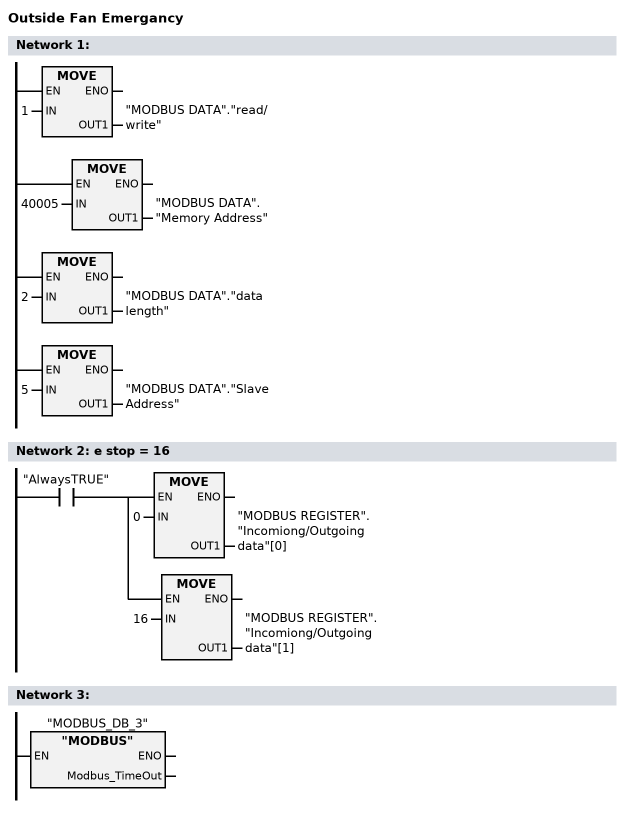
   RUNG wire#powerrail
      Move(in := 1, out1 => "MODBUS DATA"."read/write")
   END_RUNG
   RUNG wire#powerrail
      Move(in := 40005, out1 => "MODBUS DATA"."Memory Address")
   END_RUNG
   RUNG wire#powerrail
      Move(in := 2, out1 => "MODBUS DATA"."data length")
   END_RUNG
   RUNG wire#powerrail
      Move(in := 5, out1 => "MODBUS DATA"."Slave Address")
   END_RUNG
   // the same network as SCL:
   "MODBUS DATA"."read/write" := 1;
   "MODBUS DATA"."Memory Address" := 40005;
   "MODBUS DATA"."data length" := 2;
   "MODBUS DATA"."Slave Address" := 5;
END_REGION

REGION Network 2: e stop = 16
   RUNG wire#powerrail
      Contact( "AlwaysTRUE" )
      wire#w1
      Move(in := 0, out1 => "MODBUS REGISTER"."Incomiong/Outgoing data"[0])
   END_RUNG
   RUNG wire#w1
      Move(in := 16, out1 => "MODBUS REGISTER"."Incomiong/Outgoing data"[1])
   END_RUNG
   // the same network as SCL:
   IF "AlwaysTRUE" THEN
       "MODBUS REGISTER"."Incomiong/Outgoing data"[0] := 0;
       "MODBUS REGISTER"."Incomiong/Outgoing data"[1] := 16;
   END_IF;
END_REGION

REGION Network 3
   RUNG wire#powerrail
      "MODBUS_DB_3"(Modbus_TimeOut =>)
   END_RUNG
   // the same network as SCL:
   "MODBUS_DB_3"();   // "MODBUS"
END_REGION
END_FUNCTION_BLOCK

FUNCTION_BLOCK "Inside Fan Emergancy"   // FB22, LAD
{ S7_Optimized_Access := 'TRUE' }
VERSION : 0.1
BEGIN

REGION Network 1
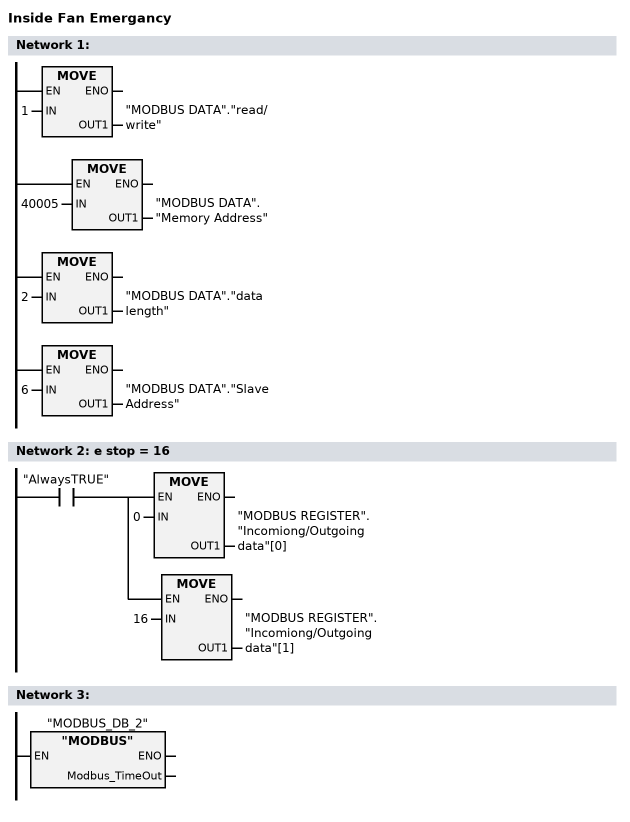
   RUNG wire#powerrail
      Move(in := 1, out1 => "MODBUS DATA"."read/write")
   END_RUNG
   RUNG wire#powerrail
      Move(in := 40005, out1 => "MODBUS DATA"."Memory Address")
   END_RUNG
   RUNG wire#powerrail
      Move(in := 2, out1 => "MODBUS DATA"."data length")
   END_RUNG
   RUNG wire#powerrail
      Move(in := 6, out1 => "MODBUS DATA"."Slave Address")
   END_RUNG
   // the same network as SCL:
   "MODBUS DATA"."read/write" := 1;
   "MODBUS DATA"."Memory Address" := 40005;
   "MODBUS DATA"."data length" := 2;
   "MODBUS DATA"."Slave Address" := 6;
END_REGION

REGION Network 2: e stop = 16
   RUNG wire#powerrail
      Contact( "AlwaysTRUE" )
      wire#w1
      Move(in := 0, out1 => "MODBUS REGISTER"."Incomiong/Outgoing data"[0])
   END_RUNG
   RUNG wire#w1
      Move(in := 16, out1 => "MODBUS REGISTER"."Incomiong/Outgoing data"[1])
   END_RUNG
   // the same network as SCL:
   IF "AlwaysTRUE" THEN
       "MODBUS REGISTER"."Incomiong/Outgoing data"[0] := 0;
       "MODBUS REGISTER"."Incomiong/Outgoing data"[1] := 16;
   END_IF;
END_REGION

REGION Network 3
   RUNG wire#powerrail
      "MODBUS_DB_2"(Modbus_TimeOut =>)
   END_RUNG
   // the same network as SCL:
   "MODBUS_DB_2"();   // "MODBUS"
END_REGION
END_FUNCTION_BLOCK

FUNCTION_BLOCK "Off Mode"   // FB23, LAD
{ S7_Optimized_Access := 'TRUE' }
VERSION : 0.1
BEGIN

REGION Network 1: Manual operation of outputs
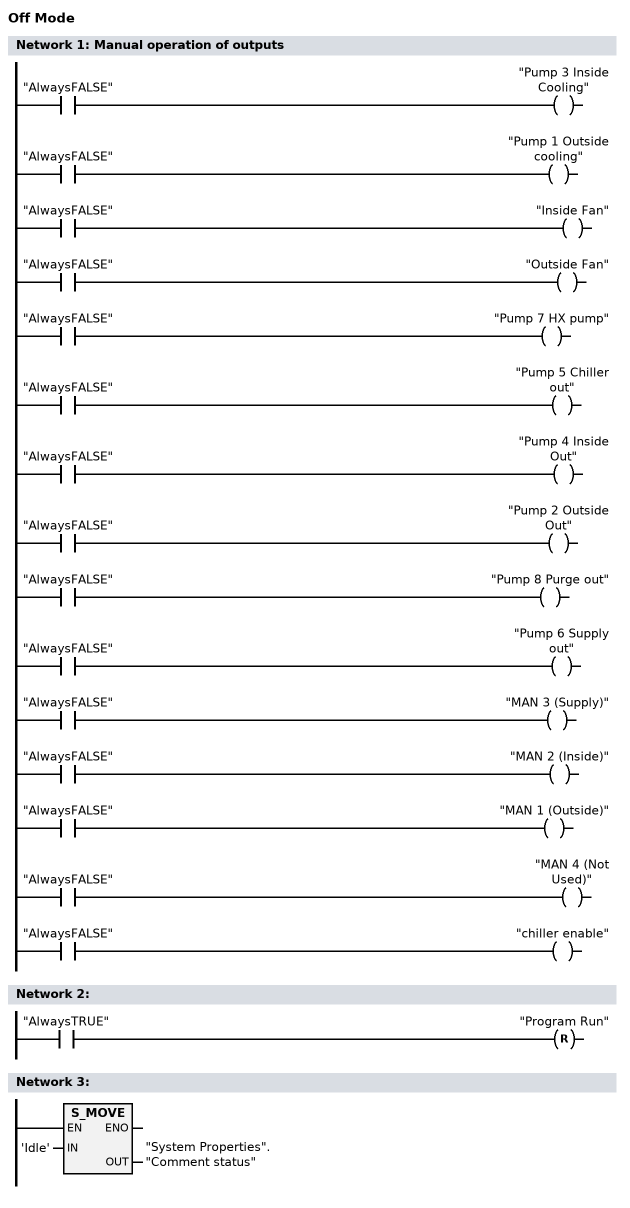
   RUNG wire#powerrail
      Contact( "AlwaysFALSE" )
      Coil( "Pump 3 Inside Cooling" )
   END_RUNG
   RUNG wire#powerrail
      Contact( "AlwaysFALSE" )
      Coil( "Pump 1 Outside cooling" )
   END_RUNG
   RUNG wire#powerrail
      Contact( "AlwaysFALSE" )
      Coil( "Inside Fan" )
   END_RUNG
   RUNG wire#powerrail
      Contact( "AlwaysFALSE" )
      Coil( "Outside Fan" )
   END_RUNG
   RUNG wire#powerrail
      Contact( "AlwaysFALSE" )
      Coil( "Pump 7 HX pump" )
   END_RUNG
   RUNG wire#powerrail
      Contact( "AlwaysFALSE" )
      Coil( "Pump 5 Chiller out" )
   END_RUNG
   RUNG wire#powerrail
      Contact( "AlwaysFALSE" )
      Coil( "Pump 4 Inside Out" )
   END_RUNG
   RUNG wire#powerrail
      Contact( "AlwaysFALSE" )
      Coil( "Pump 2 Outside Out" )
   END_RUNG
   RUNG wire#powerrail
      Contact( "AlwaysFALSE" )
      Coil( "Pump 8 Purge out" )
   END_RUNG
   RUNG wire#powerrail
      Contact( "AlwaysFALSE" )
      Coil( "Pump 6 Supply out" )
   END_RUNG
   RUNG wire#powerrail
      Contact( "AlwaysFALSE" )
      Coil( "MAN 3 (Supply)" )
   END_RUNG
   RUNG wire#powerrail
      Contact( "AlwaysFALSE" )
      Coil( "MAN 2 (Inside)" )
   END_RUNG
   RUNG wire#powerrail
      Contact( "AlwaysFALSE" )
      Coil( "MAN 1 (Outside)" )
   END_RUNG
   RUNG wire#powerrail
      Contact( "AlwaysFALSE" )
      Coil( "MAN 4 (Not Used)" )
   END_RUNG
   RUNG wire#powerrail
      Contact( "AlwaysFALSE" )
      Coil( "chiller enable" )
   END_RUNG
   // the same network as SCL:
   "Pump 3 Inside Cooling" := "AlwaysFALSE";
   "Pump 1 Outside cooling" := "AlwaysFALSE";
   "Inside Fan" := "AlwaysFALSE";
   "Outside Fan" := "AlwaysFALSE";
   "Pump 7 HX pump" := "AlwaysFALSE";
   "Pump 5 Chiller out" := "AlwaysFALSE";
   "Pump 4 Inside Out" := "AlwaysFALSE";
   "Pump 2 Outside Out" := "AlwaysFALSE";
   "Pump 8 Purge out" := "AlwaysFALSE";
   "Pump 6 Supply out" := "AlwaysFALSE";
   "MAN 3 (Supply)" := "AlwaysFALSE";
   "MAN 2 (Inside)" := "AlwaysFALSE";
   "MAN 1 (Outside)" := "AlwaysFALSE";
   "MAN 4 (Not Used)" := "AlwaysFALSE";
   "chiller enable" := "AlwaysFALSE";
END_REGION

REGION Network 2
   RUNG wire#powerrail
      Contact( "AlwaysTRUE" )
      R_Coil( "Program Run" )
   END_RUNG
   // the same network as SCL:
   IF "AlwaysTRUE" THEN "Program Run" := FALSE; END_IF;
END_REGION

REGION Network 3
   RUNG wire#powerrail
      S_Move(in := 'Idle', out => "System Properties"."Comment status")
   END_RUNG
   // the same network as SCL:
   "System Properties"."Comment status" := 'Idle';
END_REGION
END_FUNCTION_BLOCK

FUNCTION_BLOCK "Data logging main"   // FB24, LAD
{ S7_Optimized_Access := 'TRUE' }
VERSION : 0.1
BEGIN

REGION Network 1
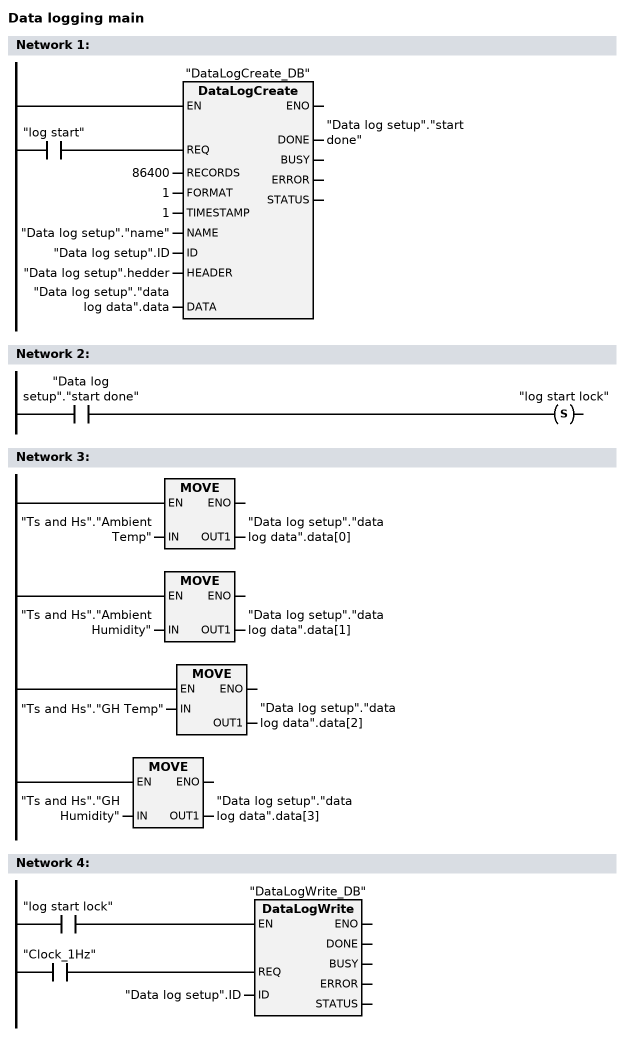
   "DataLogCreate_DB"(REQ := "log start",   // DataLogCreate
                      RECORDS := 86400,
                      FORMAT := 1,
                      TIMESTAMP := 1,
                      "NAME" := "Data log setup"."name",
                      ID := "Data log setup".ID,
                      HEADER := "Data log setup".hedder,
                      DATA := "Data log setup"."data log data".data,
                      DONE => "Data log setup"."start done");
END_REGION

REGION Network 2
   RUNG wire#powerrail
      Contact( "Data log setup"."start done" )
      S_Coil( "log start lock" )
   END_RUNG
   // the same network as SCL:
   IF "Data log setup"."start done" THEN "log start lock" := TRUE; END_IF;
END_REGION

REGION Network 3
   RUNG wire#powerrail
      Move(in := "Ts and Hs"."Ambient Temp", out1 => "Data log setup"."data log data".data[0])
   END_RUNG
   RUNG wire#powerrail
      Move(in := "Ts and Hs"."Ambient Humidity", out1 => "Data log setup"."data log data".data[1])
   END_RUNG
   RUNG wire#powerrail
      Move(in := "Ts and Hs"."GH Temp", out1 => "Data log setup"."data log data".data[2])
   END_RUNG
   RUNG wire#powerrail
      Move(in := "Ts and Hs"."GH Humidity", out1 => "Data log setup"."data log data".data[3])
   END_RUNG
   // the same network as SCL:
   "Data log setup"."data log data".data[0] := "Ts and Hs"."Ambient Temp";
   "Data log setup"."data log data".data[1] := "Ts and Hs"."Ambient Humidity";
   "Data log setup"."data log data".data[2] := "Ts and Hs"."GH Temp";
   "Data log setup"."data log data".data[3] := "Ts and Hs"."GH Humidity";
END_REGION

REGION Network 4
   IF "log start lock" THEN
       "DataLogWrite_DB"(REQ := "Clock_1Hz", ID := "Data log setup".ID);   // DataLogWrite
   END_IF;
END_REGION
END_FUNCTION_BLOCK

ORGANIZATION_BLOCK "Main"   // OB1, LAD, ProgramCycle
TITLE = "Main Program Sweep (Cycle)"
{ S7_Optimized_Access := 'TRUE' }
VERSION : 0.1
   VAR_INPUT
      Initial_Call : Bool;   // Initial call of this OB
      Remanence : Bool;   // =True, if remanent data are available
   END_VAR
   VAR_TEMP
      placeholder : Bool;
   END_VAR
   VAR_TEMP   // added for the SCL form of the ladder/FBD networks
      _w1 : Bool;
   END_VAR
BEGIN

REGION Network 1: Work out if it's day or night
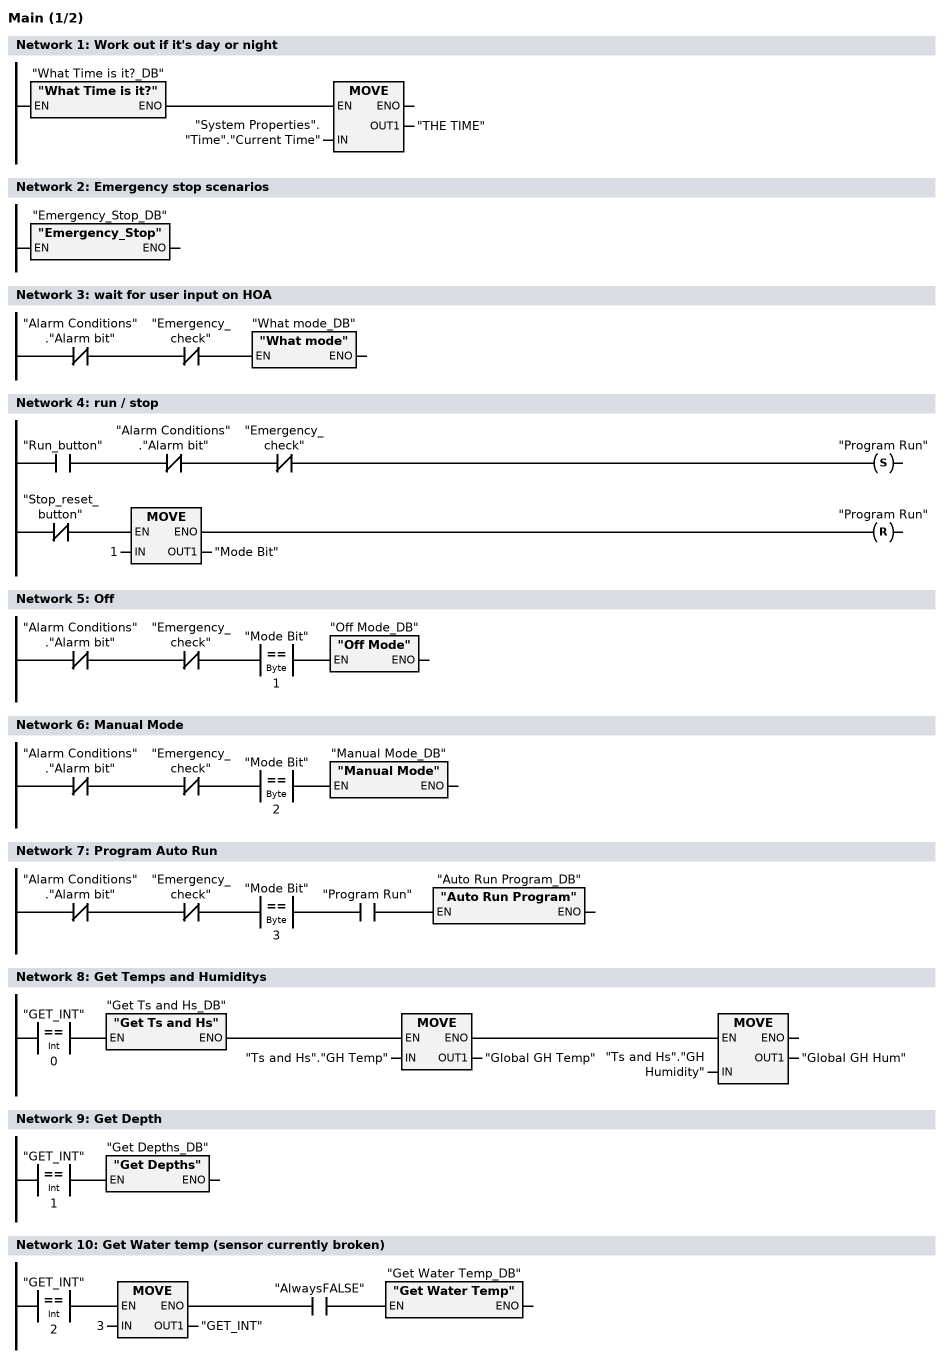
   RUNG wire#powerrail
      "What Time is it?_DB"()
      Move(in := "System Properties"."Time"."Current Time", out1 => "THE TIME")
   END_RUNG
   // the same network as SCL:
   "What Time is it?_DB"(ENO => #_w1);   // "What Time is it?"
   IF #_w1 THEN "THE TIME" := "System Properties"."Time"."Current Time"; END_IF;
END_REGION

REGION Network 2: Emergency stop scenarios
   RUNG wire#powerrail
      "Emergency_Stop_DB"()
   END_RUNG
   // the same network as SCL:
   "Emergency_Stop_DB"();   // "Emergency_Stop"
END_REGION

REGION Network 3: wait for user input on HOA
   RUNG wire#powerrail
      I_Contact( "Alarm Conditions"."Alarm bit" )
      I_Contact( "Emergency_check" )
      "What mode_DB"()
   END_RUNG
   // the same network as SCL:
   IF NOT "Alarm Conditions"."Alarm bit" AND NOT "Emergency_check" THEN
       "What mode_DB"();   // "What mode"
   END_IF;
END_REGION

REGION Network 4: run / stop
   RUNG wire#powerrail
      Contact( "Run_button" )
      I_Contact( "Alarm Conditions"."Alarm bit" )
      I_Contact( "Emergency_check" )
      S_Coil( "Program Run" )
   END_RUNG
   RUNG wire#powerrail
      I_Contact( "Stop_reset_button" )
      Move(in := 1, out1 => "Mode Bit")
      R_Coil( "Program Run" )
   END_RUNG
   // the same network as SCL:
   IF "Run_button" AND NOT "Alarm Conditions"."Alarm bit" AND NOT "Emergency_check" THEN
       "Program Run" := TRUE;
   END_IF;
   IF NOT "Stop_reset_button" THEN
       "Mode Bit" := 1;
       "Program Run" := FALSE;
   END_IF;
END_REGION

REGION Network 5: Off
   RUNG wire#powerrail
      I_Contact( "Alarm Conditions"."Alarm bit" )
      I_Contact( "Emergency_check" )
      { S7_Templates := "SrcType := Byte" } EQ_Contact(in1 := "Mode Bit", in2 := 1)
      "Off Mode_DB"()
   END_RUNG
   // the same network as SCL:
   IF NOT "Alarm Conditions"."Alarm bit" AND NOT "Emergency_check" AND ("Mode Bit" = 1) THEN
       "Off Mode_DB"();   // "Off Mode"
   END_IF;
END_REGION

REGION Network 6: Manual Mode
   RUNG wire#powerrail
      I_Contact( "Alarm Conditions"."Alarm bit" )
      I_Contact( "Emergency_check" )
      { S7_Templates := "SrcType := Byte" } EQ_Contact(in1 := "Mode Bit", in2 := 2)
      "Manual Mode_DB"()
   END_RUNG
   // the same network as SCL:
   IF NOT "Alarm Conditions"."Alarm bit" AND NOT "Emergency_check" AND ("Mode Bit" = 2) THEN
       "Manual Mode_DB"();   // "Manual Mode"
   END_IF;
END_REGION

REGION Network 7: Program Auto Run
   RUNG wire#powerrail
      I_Contact( "Alarm Conditions"."Alarm bit" )
      I_Contact( "Emergency_check" )
      { S7_Templates := "SrcType := Byte" } EQ_Contact(in1 := "Mode Bit", in2 := 3)
      Contact( "Program Run" )
      "Auto Run Program_DB"()
   END_RUNG
   // the same network as SCL:
   IF NOT "Alarm Conditions"."Alarm bit" AND NOT "Emergency_check" AND ("Mode Bit" = 3) AND "Program Run" THEN
       "Auto Run Program_DB"();   // "Auto Run Program"
   END_IF;
END_REGION

REGION Network 8: Get Temps and Humiditys
   RUNG wire#powerrail
      { S7_Templates := "SrcType := Int" } EQ_Contact(in1 := "GET_INT", in2 := 0)
      "Get Ts and Hs_DB"()
      Move(in := "Ts and Hs"."GH Temp", out1 => "Global GH Temp")
      Move(in := "Ts and Hs"."GH Humidity", out1 => "Global GH Hum")
   END_RUNG
   // the same network as SCL:
   "Get Ts and Hs_DB"(EN := "GET_INT" = 0, ENO => #_w1);   // "Get Ts and Hs"
   IF #_w1 THEN
       "Global GH Temp" := "Ts and Hs"."GH Temp";
       "Global GH Hum" := "Ts and Hs"."GH Humidity";
   END_IF;
END_REGION

REGION Network 9: Get Depth
   RUNG wire#powerrail
      { S7_Templates := "SrcType := Int" } EQ_Contact(in1 := "GET_INT", in2 := 1)
      "Get Depths_DB"()
   END_RUNG
   // the same network as SCL:
   IF "GET_INT" = 1 THEN
       "Get Depths_DB"();   // "Get Depths"
   END_IF;
END_REGION

REGION Network 10: Get Water temp (sensor currently broken)
   RUNG wire#powerrail
      { S7_Templates := "SrcType := Int" } EQ_Contact(in1 := "GET_INT", in2 := 2)
      Move(in := 3, out1 => "GET_INT")
      Contact( "AlwaysFALSE" )
      "Get Water Temp_DB"()
   END_RUNG
   // the same network as SCL:
   #_w1 := "GET_INT" = 2;
   IF #_w1 THEN "GET_INT" := 3; END_IF;
   IF #_w1 AND "AlwaysFALSE" THEN
       "Get Water Temp_DB"();   // "Get Water Temp"
   END_IF;
END_REGION

REGION Network 12: Update Inside Fans
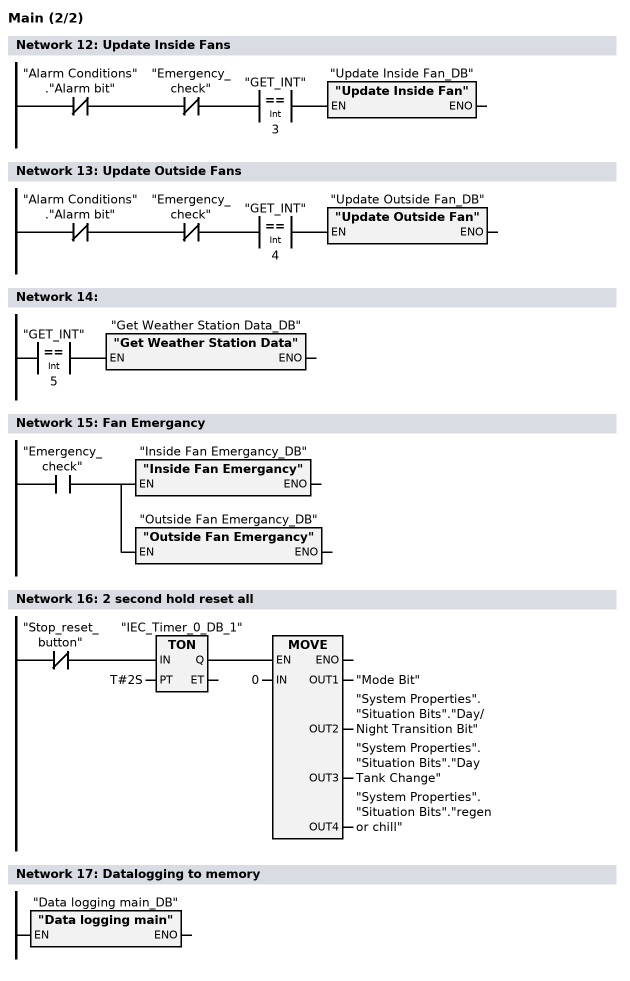
   RUNG wire#powerrail
      I_Contact( "Alarm Conditions"."Alarm bit" )
      I_Contact( "Emergency_check" )
      { S7_Templates := "SrcType := Int" } EQ_Contact(in1 := "GET_INT", in2 := 3)
      "Update Inside Fan_DB"()
   END_RUNG
   // the same network as SCL:
   IF NOT "Alarm Conditions"."Alarm bit" AND NOT "Emergency_check" AND ("GET_INT" = 3) THEN
       "Update Inside Fan_DB"();   // "Update Inside Fan"
   END_IF;
END_REGION

REGION Network 13: Update Outside Fans
   RUNG wire#powerrail
      I_Contact( "Alarm Conditions"."Alarm bit" )
      I_Contact( "Emergency_check" )
      { S7_Templates := "SrcType := Int" } EQ_Contact(in1 := "GET_INT", in2 := 4)
      "Update Outside Fan_DB"()
   END_RUNG
   // the same network as SCL:
   IF NOT "Alarm Conditions"."Alarm bit" AND NOT "Emergency_check" AND ("GET_INT" = 4) THEN
       "Update Outside Fan_DB"();   // "Update Outside Fan"
   END_IF;
END_REGION

REGION Network 14
   RUNG wire#powerrail
      { S7_Templates := "SrcType := Int" } EQ_Contact(in1 := "GET_INT", in2 := 5)
      "Get Weather Station Data_DB"()
   END_RUNG
   // the same network as SCL:
   IF "GET_INT" = 5 THEN
       "Get Weather Station Data_DB"();   // "Get Weather Station Data"
   END_IF;
END_REGION

REGION Network 15: Fan Emergancy
   RUNG wire#powerrail
      Contact( "Emergency_check" )
      wire#w1
      "Inside Fan Emergancy_DB"()
   END_RUNG
   RUNG wire#w1
      "Outside Fan Emergancy_DB"()
   END_RUNG
   // the same network as SCL:
   #_w1 := "Emergency_check";
   IF #_w1 THEN
       "Inside Fan Emergancy_DB"();   // "Inside Fan Emergancy"
       "Outside Fan Emergancy_DB"();   // "Outside Fan Emergancy"
   END_IF;
END_REGION

REGION Network 16: 2 second hold reset all
   "IEC_Timer_0_DB_1".TON(IN := NOT "Stop_reset_button", PT := T#2S);
   IF "IEC_Timer_0_DB_1".Q THEN
       "Mode Bit" := 0;
       "System Properties"."Situation Bits"."Day/Night Transition Bit" := 0;
       "System Properties"."Situation Bits"."Day Tank Change" := 0;
       "System Properties"."Situation Bits"."regen or chill" := 0;
   END_IF;
END_REGION

REGION Network 17: Datalogging to memory
   RUNG wire#powerrail
      "Data logging main_DB"()
   END_RUNG
   // the same network as SCL:
   "Data logging main_DB"();   // "Data logging main"
END_REGION
END_ORGANIZATION_BLOCK

ORGANIZATION_BLOCK "Startup"   // OB100, LAD, Startup
TITLE = "Complete Restart"
{ S7_Optimized_Access := 'TRUE' }
VERSION : 0.1
   VAR_INPUT
      LostRetentive : Bool;   // True if retentive data are lost
      LostRTC : Bool;   // True if date and time are lost
   END_VAR
   VAR_TEMP
      temp1 : Int;
      temp2 : Int;
   END_VAR
BEGIN

REGION Network 1: Put Program In Start Up Mode (0) and ensure sub program set bits are 0
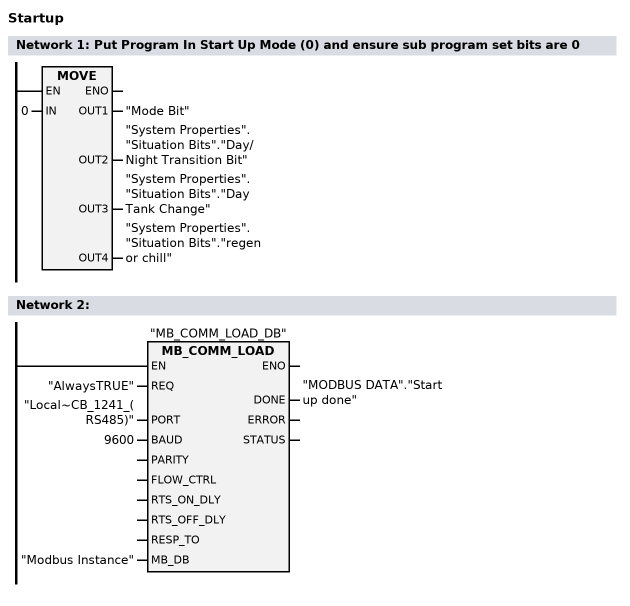
   RUNG wire#powerrail
      Move(in := 0, out1 => "Mode Bit", out2 => "System Properties"."Situation Bits"."Day/Night Transition Bit", out3 => "System Properties"."Situation Bits"."Day Tank Change", out4 => "System Properties"."Situation Bits"."regen or chill")
   END_RUNG
   // the same network as SCL:
   "Mode Bit" := 0;
   "System Properties"."Situation Bits"."Day/Night Transition Bit" := 0;
   "System Properties"."Situation Bits"."Day Tank Change" := 0;
   "System Properties"."Situation Bits"."regen or chill" := 0;
END_REGION

REGION Network 2
   "MB_COMM_LOAD_DB"(REQ := "AlwaysTRUE",   // MB_COMM_LOAD
                     PORT := "Local~CB_1241_(RS485)",
                     BAUD := 9600,
                     MB_DB := "Modbus Instance",
                     DONE => "MODBUS DATA"."Start up done");
END_REGION
END_ORGANIZATION_BLOCK

(* ===== HMI "HMI_RT_1" =====
system functions are stored by id; their names below are inferred from use

HMI tags "Default tag table"
   "Tag_ScreenNumber" : UInt, internal

Template "Template_1" 800x480
   Button "Exit" at 714,429 size 71x50; TextOff 'Exit'; PictureOff "ExitRuntime_KTP700_Basic_PN_TR"; PictureOn "ExitRuntime_KTP700_Basic_PN_TR"
      on Release: StopRuntime(0)
   Button "Template_Button" at 614,429 size 71x50; TextOff 'Text'
   Button "Template_Button_1" at 514,429 size 71x50; TextOff 'Text'
   Button "Template_Button_2" at 414,429 size 71x50; TextOff 'Text'
   Button "Template_Button_3" at 314,429 size 71x50; TextOff 'Text'
   Button "Template_Button_4" at 214,429 size 71x50; TextOff 'Text'
   Button "Template_Button_5" at 114,429 size 71x50; TextOff 'Text'
   Button "Start screen" at 14,429 size 71x50; TextOff 'Start screen'; PictureOff "NavigateHome_KTP700_Basic_PN_TR"; PictureOn "NavigateHome_KTP700_Basic_PN_TR"
      on Release: ActivateScreen("Root screen", 0)
   SymbolicIOField "Symbolic_IO_Field_Screen" at 93,9 size 600x33; TextOff '0'; TextOn '1'; TextList "TextList_ScreenNames"
      ProcessValue <- "Tag_ScreenNumber"
      on Change: ActivateScreenByNumber("Tag_ScreenNumber", 0)
   DateTimeField "HmiScreenItemData" at 695,25 size 105x25
   DateTimeField "HmiScreenItemData_1" at 695,0 size 105x25
   GraphicView "Logo" at 0,0 size 91x51; Picture "Logo of HMI_1"

screen "Root screen" 800x480, template "Template_1"
   on GenerateScreen: SetTag("Tag_ScreenNumber", 1)
   TextField "HmiScreenItemData" at 80,225 size 640x25; Text 'Welcome to HMI_1 (KTP700 Basic+ PN)!'
*)